// TIA Portal V21 export
VAR_GLOBAL   // PLC tag table "K_TipoValvola"
END_VAR
VAR_GLOBAL CONSTANT   // user constants
   K_TipoValvola_BistabileCentriChiusi : Int := 1;
   K_TipoValvola_Monostabile : Int := 0;
   K_TipoValvola_BistabileCentriAperti : Int := 2;
   K_TipoValvola_BistabileCentriApertiEChiusi : Int := 3;
   K_TipoValvola_Modulante : Int := 4;
END_VAR
